(* CODESYS project BagAdvanceMotor.xml

Project tree, tasks and I/O mapping:
  function block BagAdvanceMotor [LD]
*)

// BagAdvanceMotor
FUNCTION_BLOCK BagAdvanceMotor
// Motor: Oriental Motor Model BLM5120HP-GFV
//   	Frame Size: 90mm
// 		Output Power: 120 W
// 		Rotation Speed: 50 to 4000 r/min (Factory set to 50 r/min)
//		Torque Limiting: 0 - 300% (Factory set to 300%)
//		Acceleration and deleceration time: 0.0 to 15.0s (Factory set to 0.5s)
// Gearhead: Oriental Motor Model GFV5G30AS
// Controller: BLE2D120-A

// Motor Controller IO - Inputs map to control logic outputs, outputs map to inputs
//	1	IN-COM0	Input common for external power supplies
//	2	IN0 	FWD
//	3	IN1		REV
//	4	IN2		STOP-MODE	Select how the motor stops, when off the motor decelerates to a stop
//	5	IN3		M0			Select the desired operation data number by switching ON-OFF status of M0 and M1
//	6	IN4		M1			
//	7	IN5		ALARM-RESET
//	8	IN6		MB-FREE		Select how the brake would operate when the motor stops, if ON the brake can be released
//	9	IN-COM1	0V for external power supplies
//	10	TH		TH			
//	11	TH		TH
//	12	VH		
//	13	VM		12-14 are external analog setting input, 0-10V
//	14	VL
//	15	OUT0+	SPEED-OUT
//	16	OUT0-
//	17	OUT1+	ALARM-OUT
//	18	OUT1-

VAR_INPUT
	CommandForward: BOOL;
	CommandReverse: BOOL;
	Speed: REAL;
	Alarm: BOOL;
	ResetAlarm: BOOL;
END_VAR
VAR_OUTPUT
	Foward: BOOL;
	Reverse: BOOL;
	SpeedOutput: REAL;
	AlarmReset: BOOL;
	SpeedInputError: BOOL;
END_VAR
VAR
	MIN_SPEED: REAL := 50; // Minimum input speed in r/min
	MAX_SPEED: REAL := 4000; // Maximum input speed in r/min
	MIN_VOLTS: REAL := 0; // Minimum analog output volts
	MAX_VOLTS: REAL := 10; // Maximum analog output volts
END_VAR

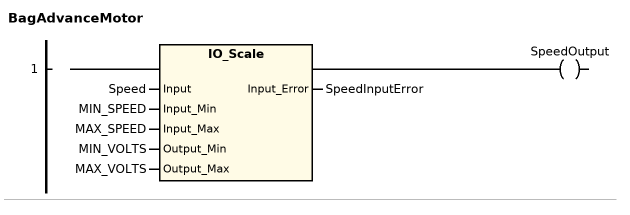
// NETWORK 1
SpeedOutput := IO_Scale(Input := Speed, Input_Min := MIN_SPEED, Input_Max := MAX_SPEED, Output_Min := MIN_VOLTS, Output_Max := MAX_VOLTS, Input_Error => SpeedInputError);

END_FUNCTION_BLOCK
